// TIA Portal V21 export
VAR_GLOBAL   // PLC tag table "K_ComunicazioneS7"
END_VAR
VAR_GLOBAL CONSTANT   // user constants
   K_ComunicazioneS7_St1_Qci : Int := 1;   // St1_qci
   K_ComunicazioneS7_St1_Robopack : Int := 2;   // St1_robopack
END_VAR
